ABB RobotStudio station: FinalProjectStation_20220130-203529.rsstn

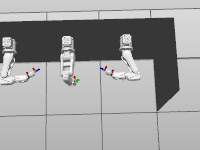
Station FinalProjectStation (saved by RobotStudio 20.4.9280.0)
Layout (positions relative to the parent item):
  - IRB120_3_58__01 [mechanism, from Robots\IRB120_3_58_G_01.rslib] at (1500, 0, 1200) mm, rotated rx 0 ry 90 rz -90 deg; joint values [0.2011, -0.2054, 0.1567, 0, 0.5236, 0] (rad or m)
  - Wall [part]
  - IRB120_3_58__01_2 [mechanism, from Robots\IRB120_3_58_G_01.rslib] at (600, 0, 1200) mm, rotated rx 0 ry 90 rz -90 deg; joint values [1.5556, -0.2111, 0.2853, 0, 0.5236, 0] (rad or m)
  - IRB120_3_58__01_3 [mechanism, from Robots\IRB120_3_58_G_01.rslib] at (2400, 0, 1200) mm, rotated rx 0 ry 90 rz -90 deg; joint values [-1.5848, -0.4515, 0.4678, 0, 0.5236, 0] (rad or m)
  - Smart_Gripper_Servo_Fingers [mechanism, from Tools\ABB_Smart_Gripper_Servo_Fingers.rslib] at (1561.37, -605.99, 898.98) mm, rotated rx 167.09 ry -26.62 rz 95.87 deg; joint values [0] (rad or m)
  - Smart_Gripper_Servo_Fingers_2 [mechanism, from Tools\ABB_Smart_Gripper_Servo_Fingers.rslib] at (909.26, -560.91, 1195.3) mm, rotated rx 90.72 ry -0.49 rz 124.25 deg; joint values [0] (rad or m)
  - Smart_Gripper_Servo_Fingers_3 [mechanism, from Tools\ABB_Smart_Gripper_Servo_Fingers.rslib] at (2152.97, -561.01, 1203.47) mm, rotated rx -89.31 ry 0.41 rz 59.07 deg; joint values [0] (rad or m)
Attachment: Smart_Gripper_Servo_Fingers is attached to IRB120_3_58__01 / Link6
Attachment: Smart_Gripper_Servo_Fingers_2 is attached to IRB120_3_58__01_2 / Link6
Attachment: Smart_Gripper_Servo_Fingers_3 is attached to IRB120_3_58__01_3 / Link6
Targets, tools, work objects and paths stored in the station, written as RAPID:
! task (no controller)
MODULE CalibData
  PERS tooldata Servo:=[TRUE,[[0,0,114.2],[1,0,0,0]],[0.215,[8.7,12.3,49.2],[1,0,0,0],0.00021,0.00024,0.00009]];
ENDMODULE

! task (no controller)
MODULE CalibData
  PERS tooldata Servo:=[TRUE,[[0,0,114.2],[1,0,0,0]],[0.215,[8.7,12.3,49.2],[1,0,0,0],0.00021,0.00024,0.00009]];
ENDMODULE

! task (no controller)
MODULE CalibData
  PERS tooldata Servo:=[TRUE,[[0,0,114.2],[1,0,0,0]],[0.215,[8.7,12.3,49.2],[1,0,0,0],0.00021,0.00024,0.00009]];
ENDMODULE

